// TIA Portal V20 export
FUNCTION "EM2_TeachingData" : Void   // FC73, FBD
// stored: Namespace Unit1.Em2, SetENOAutomatically false
BEGIN

REGION Network 2 (SCL): JROutPnP Left AxisX Teaching Position
   //JROutPnPLeft AxisX Position 0
   "Unit1.Em2.HmiInterface".cmJROutPnPLeftAxisX.configuration.setPositions[0].position := 4273.91;
   "Unit1.Em2.HmiInterface".cmJROutPnPLeftAxisX.configuration.setPositions[0].velocity := 50.0;

   //JROutPnPLeft AxisX Position 1
   "Unit1.Em2.HmiInterface".cmJROutPnPLeftAxisX.configuration.setPositions[1].position := -9.0;
   "Unit1.Em2.HmiInterface".cmJROutPnPLeftAxisX.configuration.setPositions[1].velocity := 50.0;

   //JROutPnPLeft AxisX Position 2
   "Unit1.Em2.HmiInterface".cmJROutPnPLeftAxisX.configuration.setPositions[2].position := 3402.93;
   "Unit1.Em2.HmiInterface".cmJROutPnPLeftAxisX.configuration.setPositions[2].velocity := 50.0;

   //JROutPnPLeft AxisX Position 3
   "Unit1.Em2.HmiInterface".cmJROutPnPLeftAxisX.configuration.setPositions[3].position := 4825.92;
   "Unit1.Em2.HmiInterface".cmJROutPnPLeftAxisX.configuration.setPositions[3].velocity := 50.0;


   ///////////////////////////////////// Zone ///////////////////////////

   //JROutPnPLeft AxisX Position 8
   "Unit1.Em2.HmiInterface".cmJROutPnPLeftAxisX.configuration.setPositions[8].position := 1700.0;
   "Unit1.Em2.HmiInterface".cmJROutPnPLeftAxisX.configuration.setPositions[8].velocity := 50.0;

   //JROutPnPLeft AxisX Position 9
   "Unit1.Em2.HmiInterface".cmJROutPnPLeftAxisX.configuration.setPositions[9].position := -9.0;
   "Unit1.Em2.HmiInterface".cmJROutPnPLeftAxisX.configuration.setPositions[9].velocity := 50.0;

   //JROutPnPLeft AxisX Position 10
   "Unit1.Em2.HmiInterface".cmJROutPnPLeftAxisX.configuration.setPositions[10].position := 3402.93;
   "Unit1.Em2.HmiInterface".cmJROutPnPLeftAxisX.configuration.setPositions[10].velocity := 50.0;

   //JROutPnPLeft AxisX Position 11
   "Unit1.Em2.HmiInterface".cmJROutPnPLeftAxisX.configuration.setPositions[11].position := 4825.92;
   "Unit1.Em2.HmiInterface".cmJROutPnPLeftAxisX.configuration.setPositions[11].velocity := 50.0;
END_REGION

REGION Network 3 (SCL): JROutPnP Left AxisZ Teeaching Position
   // JROutPnPLeft AxisZ Position 0
   "Unit1.Em2.HmiInterface".cmJROutPnPLeftAxisZ.configuration.setPositions[0].position := 0.0;
   "Unit1.Em2.HmiInterface".cmJROutPnPLeftAxisZ.configuration.setPositions[0].velocity := 10.0;

   // JROutPnPLeft AxisZ Position 1
   "Unit1.Em2.HmiInterface".cmJROutPnPLeftAxisZ.configuration.setPositions[1].position := 356.0;
   "Unit1.Em2.HmiInterface".cmJROutPnPLeftAxisZ.configuration.setPositions[1].velocity := 10.0;

   // JROutPnPLeft AxisZ Position 2
   "Unit1.Em2.HmiInterface".cmJROutPnPLeftAxisZ.configuration.setPositions[2].position := 356.0;
   "Unit1.Em2.HmiInterface".cmJROutPnPLeftAxisZ.configuration.setPositions[2].velocity := 10.0;

   // JROutPnPLeft AxisZ Position 3
   "Unit1.Em2.HmiInterface".cmJROutPnPLeftAxisZ.configuration.setPositions[3].position := 329.0;
   "Unit1.Em2.HmiInterface".cmJROutPnPLeftAxisZ.configuration.setPositions[3].velocity := 10.0;


   ///////////////////////////////////// Zone ///////////////////////////

   // JROutPnPLeft AxisZ Position 8
   "Unit1.Em2.HmiInterface".cmJROutPnPLeftAxisZ.configuration.setPositions[8].position := 0.0;
   "Unit1.Em2.HmiInterface".cmJROutPnPLeftAxisZ.configuration.setPositions[8].velocity := 10.0;
END_REGION

REGION Network 4 (SCL): JROutPnP Right AxisX Teaching Position
   //JROutPnPRight AxisX Position 0
   "Unit1.Em2.HmiInterface".cmJROutPnPRightAxisX.configuration.setPositions[0].position := 600.0;
   "Unit1.Em2.HmiInterface".cmJROutPnPRightAxisX.configuration.setPositions[0].velocity := 50.0;

   //JROutPnPRight AxisX Position 1
   "Unit1.Em2.HmiInterface".cmJROutPnPRightAxisX.configuration.setPositions[1].position := 1277.8;
   "Unit1.Em2.HmiInterface".cmJROutPnPRightAxisX.configuration.setPositions[1].velocity := 50.0;

   //JROutPnPRight AxisX Position 2
   "Unit1.Em2.HmiInterface".cmJROutPnPRightAxisX.configuration.setPositions[2].position := 5.0;
   "Unit1.Em2.HmiInterface".cmJROutPnPRightAxisX.configuration.setPositions[2].velocity := 50.0;


   ///////////////////////////////////// Zone ///////////////////////////

   //JROutPnPRight AxisX Position 8
   "Unit1.Em2.HmiInterface".cmJROutPnPRightAxisX.configuration.setPositions[8].position := 600.0;
   "Unit1.Em2.HmiInterface".cmJROutPnPRightAxisX.configuration.setPositions[8].velocity := 50.0;

   //JROutPnPRight AxisX Position 9
   "Unit1.Em2.HmiInterface".cmJROutPnPRightAxisX.configuration.setPositions[9].position := 1277.8;
   "Unit1.Em2.HmiInterface".cmJROutPnPRightAxisX.configuration.setPositions[9].velocity := 50.0;

   //JROutPnPRight AxisX Position 10
   "Unit1.Em2.HmiInterface".cmJROutPnPRightAxisX.configuration.setPositions[10].position := 5.0;
   "Unit1.Em2.HmiInterface".cmJROutPnPRightAxisX.configuration.setPositions[10].velocity := 50.0;
END_REGION

REGION Network 5 (SCL): JROutPnP Right AxisZ Teeaching Position
   // JROutPnPRight AxisZ Position 0
   "Unit1.Em2.HmiInterface".cmJROutPnPRightAxisZ.configuration.setPositions[0].position := 16.86;
   "Unit1.Em2.HmiInterface".cmJROutPnPRightAxisZ.configuration.setPositions[0].velocity := 10.0;

   // JROutPnPRight AxisZ Position 1
   "Unit1.Em2.HmiInterface".cmJROutPnPRightAxisZ.configuration.setPositions[1].position := 16.86;
   "Unit1.Em2.HmiInterface".cmJROutPnPRightAxisZ.configuration.setPositions[1].velocity := 10.0;

   // JROutPnPRight AxisZ Position 2
   "Unit1.Em2.HmiInterface".cmJROutPnPRightAxisZ.configuration.setPositions[2].position := 480.0;
   "Unit1.Em2.HmiInterface".cmJROutPnPRightAxisZ.configuration.setPositions[2].velocity := 10.0;

   // JROutPnPRight AxisZ Position 3
   "Unit1.Em2.HmiInterface".cmJROutPnPRightAxisZ.configuration.setPositions[3].position := 329.0;
   "Unit1.Em2.HmiInterface".cmJROutPnPRightAxisZ.configuration.setPositions[3].velocity := 10.0;


   ///////////////////////////////////// Zone ///////////////////////////

   // JROutPnPRight AxisZ Position 8
   "Unit1.Em2.HmiInterface".cmJROutPnPRightAxisZ.configuration.setPositions[8].position := 0.0;
   "Unit1.Em2.HmiInterface".cmJROutPnPRightAxisZ.configuration.setPositions[8].velocity := 10.0;
END_REGION
END_FUNCTION
